// TIA Portal V21 export
VAR_GLOBAL   // PLC tag table "PastorizzatoreSendDigitali"
END_VAR
VAR_GLOBAL CONSTANT   // user constants
   K_SegnaleVersoPastorizzatore_Marcia : Int := 1;
END_VAR
